// TIA Portal project "FactoryIO_Template_S7-1200_V15_V15.1" (V15.1)
// Vorlageprojekt für das Buch mit Zielsystem S7-1200

(* hardware
DEVICE "S7-1200-Station_1"  S7-1200 Station
   slot 0: "Baugruppenträger_0"  Rack  V1.0
   slot 1: "PLC_1"  CPU 1211C DC/DC/DC  6ES7 211-1AE40-0XB0  V4.1
DEVICE "HMI_1"  KTP900 Basic PN
   slot 0: "HMI_1"  KTP900 Basic PN  6AV2 123-2JB03-0AX0  15.1.0.0
   slot 1: "HMI_RT_1"  KTP900 Basic PN  6AV2 123-2JB03-0AX0  15.1.0.0
   slot 5: "HMI_1.IE_CP_1"  PROFINET Interface  15.0.1.0
      slot 1: "PROFINET Interface_1"  PROFINET Interface
         slot 1: "Port_1"  Port
*)

// ===== PLC "PLC_1"  CPU 1211C DC/DC/DC =====

VAR_GLOBAL   // PLC tag table "Standard-Variablentabelle"
   "Conv_1" AT %A0.0 : Bool;
   "Item_ready" AT %E0.0 : Bool;
   "At_entry" AT %E0.1 : Bool;
   "Conv_2" AT %Q0.1 : Bool;
   "At_exit" AT %I0.2 : Bool;
   "running" AT %I0.3 : Bool;
   "emitter" AT %Q0.2 : Bool;
   "Clock_Byte" AT %MB0 : Byte;
   "Clock_10Hz" AT %M0.0 : Bool;
   "Clock_5Hz" AT %M0.1 : Bool;
   "Clock_2.5Hz" AT %M0.2 : Bool;
   "Clock_2Hz" AT %M0.3 : Bool;
   "Clock_1.25Hz" AT %M0.4 : Bool;
   "Clock_1Hz" AT %M0.5 : Bool;
   "Clock_0.625Hz" AT %M0.6 : Bool;
   "Clock_0.5Hz" AT %M0.7 : Bool;
END_VAR

DATA_BLOCK "Auxiliare"   // DB1
{ S7_Optimized_Access := 'TRUE' }
VERSION : 0.1
   VAR
      nr_cutii_cerut : USInt;
      nr_cutii_curent : USInt;
      comanda_Start : Bool;
      re1 : Bool;
   END_VAR
BEGIN
END_DATA_BLOCK

FUNCTION "MHJ-PLC-Lab-Function-S71200" : Void   // FC9000, SCL
{ S7_Optimized_Access := 'TRUE' }
VERSION : 0.1
   VAR_TEMP
      rdTimeReturn : Int;
      outputTime : DTL;
      SyncVal : Byte;
      forVal : Int;
      forVal_2 : Int;
      Value : Byte;
   END_VAR
   VAR CONSTANT
      CompVal : Byte := 16#34;
      Value_01 : Byte := 16#11;
      Value_01_DW : DWord := 16#A165_D992;
      Value_02_DW : DWord := 16#58BE_4401;
   END_VAR
BEGIN

   #Value:=PEEK(area := 16#82,
        dbNumber := 0,
        byteOffset := 511);
   #Value := #Value + 1;

   POKE(area := 16#82,
        dbNumber := 0,
        byteOffset := 511,
        value := #Value);

   POKE(area:=16#81,
        dbNumber:=0,
        byteOffset:=1016,
        value:=#Value_01_DW);
   POKE(area := 16#81,
        dbNumber := 0,
        byteOffset := 1020,
        value := #Value_02_DW);

   POKE(area := 16#81,
        dbNumber := 0,
        byteOffset := 511,
        value := B#16#00);

   FOR #forVal := 0 TO 120 DO
       FOR #forVal_2:=0 TO 10 DO
           #rdTimeReturn:=RD_SYS_T(#outputTime);
           #rdTimeReturn := WR_SYS_T(#outputTime);
           #rdTimeReturn := RD_SYS_T(#outputTime);
           #rdTimeReturn := WR_SYS_T(#outputTime);
       END_FOR;
       #SyncVal:= PEEK(area := 16#81,
                      dbNumber := 0,
                      byteOffset := 511);
       IF #SyncVal = #CompVal THEN
          GOTO M_1;
       END_IF;
   END_FOR;
   RETURN;

   M_1:
   POKE(area := 16#81,
        dbNumber := 0,
        byteOffset := 511,
        value := B#16#0);
END_FUNCTION

ORGANIZATION_BLOCK "Main"   // OB1, LAD, ProgramCycle
TITLE = "Main Program Sweep (Cycle)"
{ S7_Optimized_Access := 'TRUE' }
VERSION : 0.1
   VAR_INPUT
      Initial_Call : Bool;   // Initial call of this OB
      Remanence : Bool;   // =True, if remanent data are available
   END_VAR
   VAR_TEMP   // added for the SCL form of the ladder/FBD networks
      _w1 : Bool;
   END_VAR
BEGIN

REGION Network 1: Konnektierungsbaustein für PLC-Lab
   // Im Netzwerk 1 wird der Konnektierungsbaustein für PLC-Lab aufgerufen.
   // Dieser Aufruf darf nicht entfernt werden!
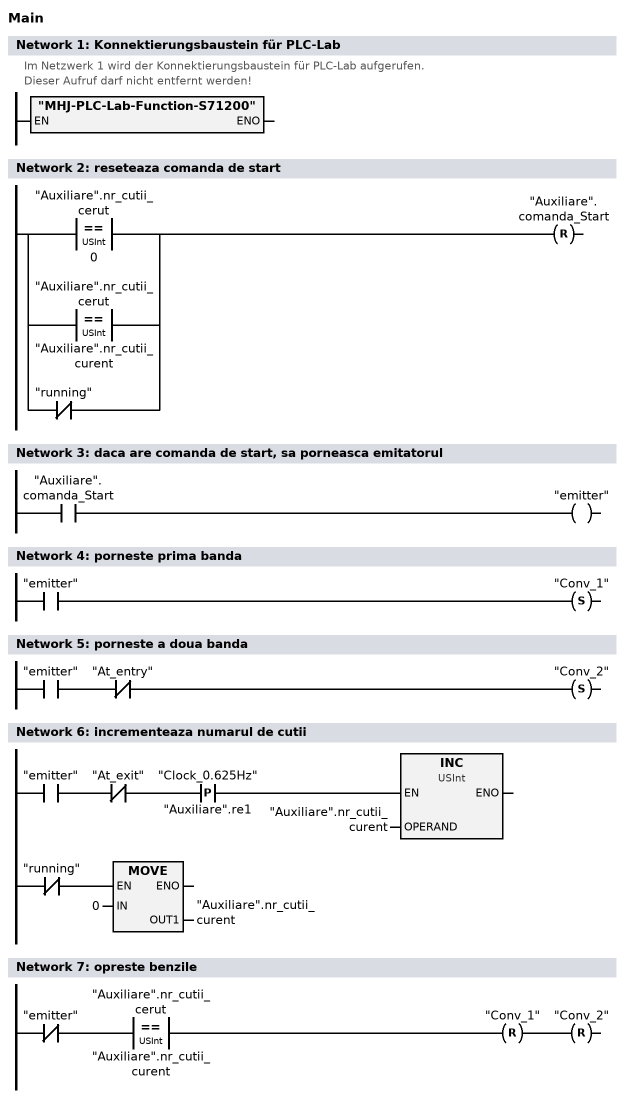
   RUNG wire#powerrail
      "MHJ-PLC-Lab-Function-S71200"()
   END_RUNG
   // the same network as SCL:
   "MHJ-PLC-Lab-Function-S71200"();
END_REGION

REGION Network 2: reseteaza comanda de start
   RUNG wire#powerrail
      { S7_Templates := "SrcType := USInt" } EQ_Contact(in1 := "Auxiliare".nr_cutii_cerut, in2 := 0)
      wire#w1
      R_Coil( "Auxiliare".comanda_Start )
   END_RUNG
   RUNG wire#powerrail
      { S7_Templates := "SrcType := USInt" } EQ_Contact(in1 := "Auxiliare".nr_cutii_cerut, in2 := "Auxiliare".nr_cutii_curent)
   END_RUNG wire#w1
   RUNG wire#powerrail
      I_Contact( "running" )
   END_RUNG wire#w1
   // the same network as SCL:
   IF ("Auxiliare".nr_cutii_cerut = 0) OR ("Auxiliare".nr_cutii_cerut = "Auxiliare".nr_cutii_curent) OR NOT "running" THEN
       "Auxiliare".comanda_Start := FALSE;
   END_IF;
END_REGION

REGION Network 3: daca are comanda de start, sa porneasca emitatorul
   RUNG wire#powerrail
      Contact( "Auxiliare".comanda_Start )
      Coil( "emitter" )
   END_RUNG
   // the same network as SCL:
   "emitter" := "Auxiliare".comanda_Start;
END_REGION

REGION Network 4: porneste prima banda
   RUNG wire#powerrail
      Contact( "emitter" )
      S_Coil( "Conv_1" )
   END_RUNG
   // the same network as SCL:
   IF "emitter" THEN "Conv_1" := TRUE; END_IF;
END_REGION

REGION Network 5: porneste a doua banda
   RUNG wire#powerrail
      Contact( "emitter" )
      I_Contact( "At_entry" )
      S_Coil( "Conv_2" )
   END_RUNG
   // the same network as SCL:
   IF "emitter" AND NOT "At_entry" THEN "Conv_2" := TRUE; END_IF;
END_REGION

REGION Network 6: incrementeaza numarul de cutii
   RUNG wire#powerrail
      Contact( "emitter" )
      I_Contact( "At_exit" )
      P_Contact(operand := "Clock_0.625Hz", bit := "Auxiliare".re1)
      { S7_Templates := "DestType := USInt" } Inc( "Auxiliare".nr_cutii_curent )
   END_RUNG
   RUNG wire#powerrail
      I_Contact( "running" )
      Move(in := 0, out1 => "Auxiliare".nr_cutii_curent)
   END_RUNG
   // the same network as SCL:
   #_w1 := "emitter" AND NOT "At_exit" AND "Clock_0.625Hz" AND NOT "Auxiliare".re1;   // rising edge of "Clock_0.625Hz"
   "Auxiliare".re1 := "Clock_0.625Hz";
   IF #_w1 THEN "Auxiliare".nr_cutii_curent := "Auxiliare".nr_cutii_curent + 1; END_IF;
   IF NOT "running" THEN "Auxiliare".nr_cutii_curent := 0; END_IF;
END_REGION

REGION Network 7: opreste benzile
   RUNG wire#powerrail
      I_Contact( "emitter" )
      { S7_Templates := "SrcType := USInt" } EQ_Contact(in1 := "Auxiliare".nr_cutii_cerut, in2 := "Auxiliare".nr_cutii_curent)
      R_Coil( "Conv_1" )
      R_Coil( "Conv_2" )
   END_RUNG
   // the same network as SCL:
   IF NOT "emitter" AND ("Auxiliare".nr_cutii_cerut = "Auxiliare".nr_cutii_curent) THEN
       "Conv_1" := FALSE;
       "Conv_2" := FALSE;
   END_IF;
END_REGION

REGION Network 8: opreste banda 2
END_REGION
END_ORGANIZATION_BLOCK

(* ===== HMI "HMI_RT_1" =====
system functions are stored by id; their names below are inferred from use
connection "HMI_Connection_1": ETHERNET, SMART_S7_1200_OMS

HMI tags "Default tag table"
   "Fill" : Bool = PLC Item_ready AT %I0.0, 1 s
   "Discharge" : Bool = PLC At_entry AT %I0.1, 1 s
   "running" : Bool = PLC running AT %I0.3, 1 s
   "Auxiliare_nr_cutii_cerut" : USInt = PLC Auxiliare.nr_cutii_cerut, 1 s
   "Auxiliare_comanda_Start" : Bool = PLC Auxiliare.comanda_Start, 1 s
   "Auxiliare_nr_cutii_curent" : USInt = PLC Auxiliare.nr_cutii_curent, 1 s

Template "Template_1" 800x480
   Button "Exit" at 722,440 size 55x39; TextOff 'Exit'; PictureOff "ExitRuntime_KTP900_Basic_PN_TR"; PictureOn "ExitRuntime_KTP900_Basic_PN_TR"
      on Release: StopRuntime(0)
   Button "Template_Button" at 622,440 size 55x39; TextOff 'Text'
   Button "Template_Button_1" at 522,440 size 55x39; TextOff 'Text'
   Button "Template_Button_2" at 422,440 size 55x39; TextOff 'Text'
   Button "Template_Button_3" at 322,440 size 55x39; TextOff 'Text'
   Button "Template_Button_4" at 222,440 size 55x39; TextOff 'Text'
   Button "Template_Button_5" at 122,440 size 55x39; TextOff 'Text'
   Button "Start screen" at 22,440 size 55x39; TextOff 'Start screen'; PictureOff "NavigateHome_KTP900_Basic_PN_TR"; PictureOn "NavigateHome_KTP900_Basic_PN_TR"
      on Release: ActivateScreen("Main", 0)

screen "Main" 800x480, template "Template_1"
   IOField "I/O field_1" at 349,112 size 102x43; FormatPattern 999
      ProcessValue <- "Auxiliare_nr_cutii_cerut"
   TextField "Text field_1" at 369,83 size 62x20; Text 'Nr. cerut'
   Button "Button_1" at 349,176 size 102x38; TextOff 'Pornire'
      on Click: SetBit("Auxiliare_comanda_Start")
   Circle "Circle_1" at 372,230 size 56x56
      Appearance <- "running"
   IOField "I/O field_2" at 352,328 size 96x32; FormatPattern 999
      ProcessValue <- "Auxiliare_nr_cutii_curent"
   TextField "Text field_2" at 366,299 size 70x20; Text 'Nr. curent'
*)